% RSLogix 500 project P6_IVANOVSKI_M.RSS, saved by version 8.30.00.16 %
PROJECT "UNTITLED"    % processor: Bul.1763 MicroLogix 1100 Series B %

PROGRAM FILES
  LAD 2 "MAIN"  3 rungs
  LAD 3 "IO"  2 rungs
  LAD 4 "HRMETER"  8 rungs

DATA FILES
  O0 OUTPUT  4 elements
  I1 INPUT  6 elements
  S2 STATUS  66 elements
  B3 BINARY  2 elements
  T4 TIMER  3 elements
  C5 COUNTER  3 elements
  R6 CONTROL  1 elements
  N7 INTEGER  4 elements
  F8 FLOAT  1 elements

LADDER 2 "MAIN"
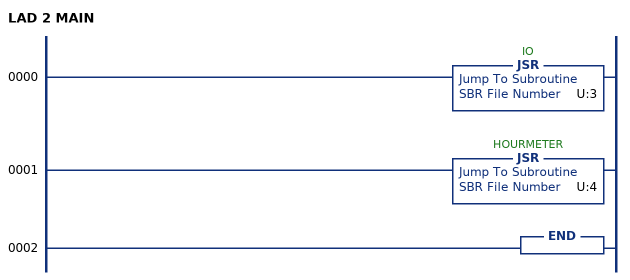
% Rung: 0 %
SOR JSR U:3 EOR
%   U:3  "IO" %
% Rung: 1 %
SOR JSR U:4 EOR
%   U:4  "HOURMETER" %
% Rung: 2 %
SOR END EOR

LADDER 3 "IO"
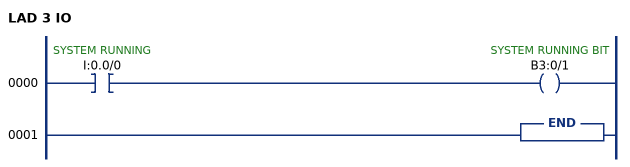
% Rung: 0 %
SOR XIC I:0.0/0 OTE B3:0/1 EOR
%   I:0.0/0  "SYSTEM RUNNING" %
%   B3:0/1  "SYSTEM RUNNING BIT" %
% Rung: 1 %
SOR END EOR

LADDER 4 "HRMETER"
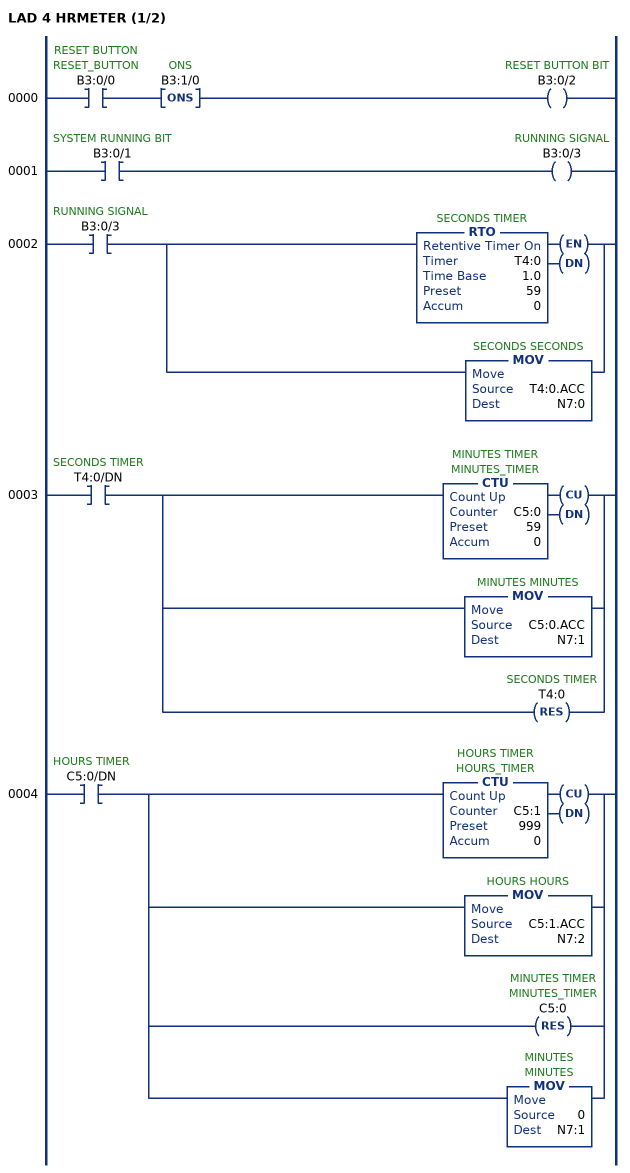
% Rung: 0 %
SOR XIC B3:0/0 ONS B3:1/0 OTE B3:0/2 EOR
%   B3:0/0  RESET_BUTTON  "RESET BUTTON" %
%   B3:1/0  "ONS" %
%   B3:0/2  "RESET BUTTON BIT" %
% Rung: 1 %
SOR XIC B3:0/1 OTE B3:0/3 EOR
%   B3:0/1  "SYSTEM RUNNING BIT" %
%   B3:0/3  "RUNNING SIGNAL" %
% Rung: 2 %
SOR XIC B3:0/3 BST RTO T4:0 1.0 59 0 NXB MOV T4:0.ACC N7:0 BND EOR
%   B3:0/3  "RUNNING SIGNAL" %
%   T4:0  "SECONDS TIMER" %
%   T4:0.ACC  "SECONDS ACCUMULATED" %
%   N7:0  SECONDS  "SECONDS" %
% Rung: 3 %
SOR XIC T4:0/DN BST CTU C5:0 59 0 NXB MOV C5:0.ACC N7:1 NXB RES T4:0 BND EOR
%   T4:0/DN  "SECONDS TIMER" %
%   C5:0  MINUTES_TIMER  "MINUTES TIMER" %
%   C5:0.ACC  "MINUTES COUNTER" %
%   N7:1  MINUTES  "MINUTES" %
%   T4:0  "SECONDS TIMER" %
% Rung: 4 %
SOR XIC C5:0/DN BST CTU C5:1 999 0 NXB MOV C5:1.ACC N7:2 NXB RES C5:0 NXB MOV 0 N7:1 BND EOR
%   C5:0/DN  "HOURS TIMER" %
%   C5:1  HOURS_TIMER  "HOURS TIMER" %
%   C5:1.ACC  "HOURS TIMER" %
%   N7:2  HOURS  "HOURS" %
%   C5:0  MINUTES_TIMER  "MINUTES TIMER" %
%   N7:1  MINUTES  "MINUTES" %

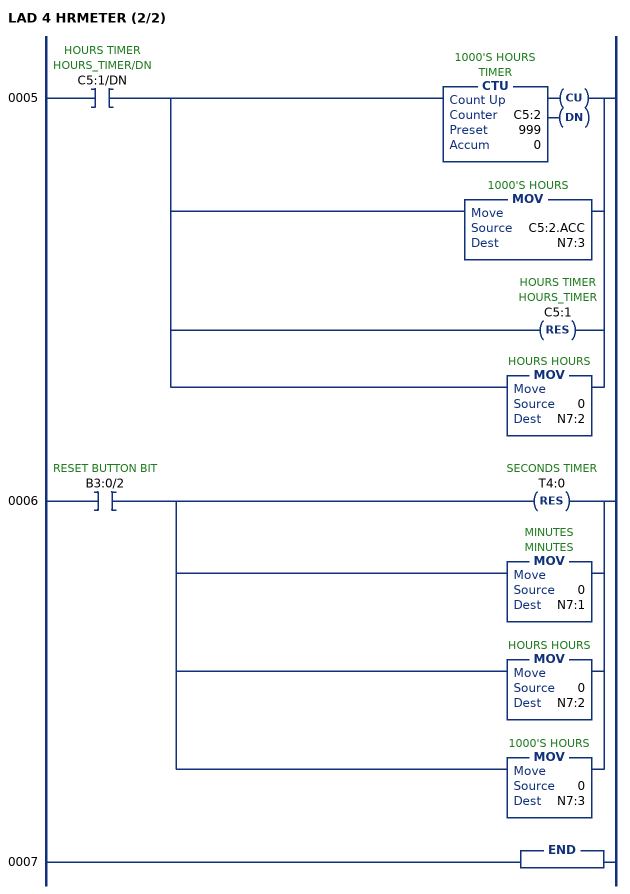
% Rung: 5 %
SOR XIC C5:1/DN BST CTU C5:2 999 0 NXB MOV C5:2.ACC N7:3 NXB RES C5:1 NXB MOV 0 N7:2 BND EOR
%   C5:1  HOURS_TIMER  "HOURS TIMER" %
%   C5:2  "1000'S HOURS TIMER" %
%   C5:2.ACC  "1000'S HOURS COUNTER" %
%   N7:3  "1000'S HOURS" %
%   N7:2  HOURS  "HOURS" %
% Rung: 6 %
SOR XIC B3:0/2 BST RES T4:0 NXB MOV 0 N7:1 NXB MOV 0 N7:2 NXB MOV 0 N7:3 BND EOR
%   B3:0/2  "RESET BUTTON BIT" %
%   T4:0  "SECONDS TIMER" %
%   N7:1  MINUTES  "MINUTES" %
%   N7:2  HOURS  "HOURS" %
%   N7:3  "1000'S HOURS" %
% Rung: 7 %
SOR END EOR

OTHER DOCUMENTED ADDRESSES
  T4:1  "MINUTES TIMER"
  T4:2  "HOURS TIMER"

DATA TABLE (non-zero values as saved)
DATA T4
% .PRE .ACC %
% T4:0 % 59 0
% T4:1 % 59 0
% T4:2 % 999 0
DATA C5
% .PRE .ACC %
% C5:0 % 59 0
% C5:1 % 999 0
% C5:2 % 999 0
